RoboDK station: 01A - Rectangle.rdk

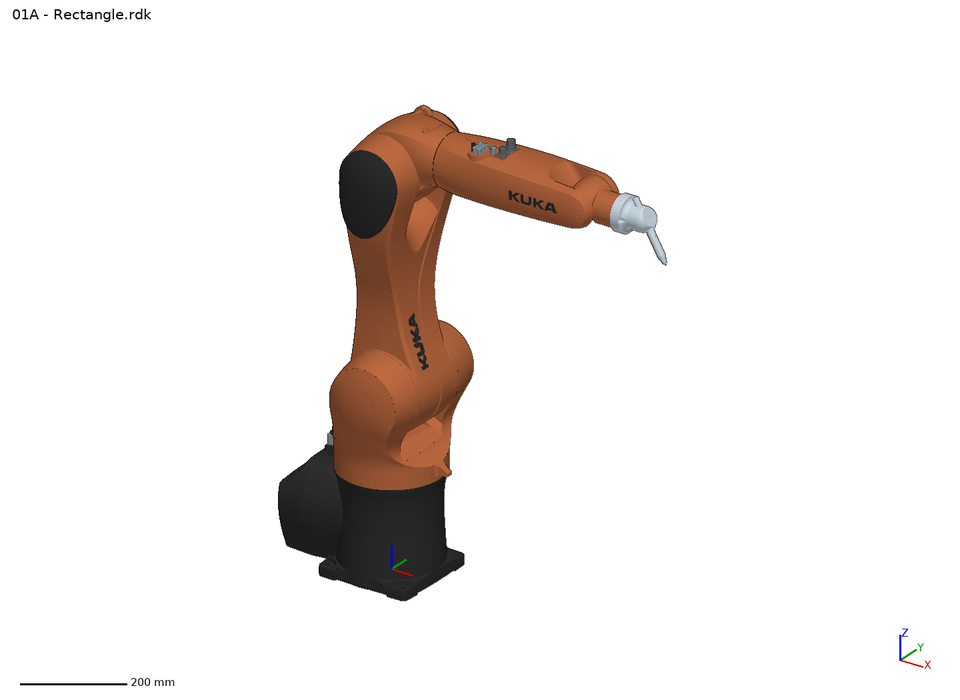
[picture v0: the station drawn from its stored meshes, robots at their saved joint values, targets as dots, program paths as lines]
Station 01A - Rectangle (saved by RoboDK 5.2.3). Poses are relative to the parent item; angles as X-Y-Z fixed-axis rotations.
Station parameters (name, value as stored): Palletizing Plugin
  - frame KUKA KR 6 R900 sixx Base at (0, 0, 0) mm
    - robot KUKA KR 6 R900 sixx: 6 axes, payload 6 kg, reach 901 mm, repeatability 0.03 mm, weight 52 kg
        modified DH rows (alpha deg, a mm, theta deg, d mm): 0, 0, 0, 400; -90, 25, 0, 0; 0, 455, -90, 0; -90, 35, 0, 420; 90, 0, 0, 0; -90, 0, 180, 80
        joint limits [-170, -190, -120, -185, -120, -350] to [170, 45, 156, 185, 120, 350]; home [0, -90, 90, 0, 0, 0]; saved at [0, -90, 90, 0, 0, 0]
      - tool Pencil, TCP at (82.67, 0, 101.52) mm, rotated rx 0 ry 60 rz 0 deg, size 125 x 74.9 x 107.3 mm
